{attribute 'TcGenerated'}
{attribute 'no-analysis'}
{attribute 'linkalways'}
// This function has been automatically generated from the project information.
VAR_GLOBAL CONSTANT
	{attribute 'const_non_replaced'}
	stLibVersion_Intecre_File : ST_LibVersion := (iMajor := 0, iMinor := 2, iBuild := 0, iRevision := 0, sVersion := '0.2.0');
END_VAR

(* stored: Version 1.1.0.1, ProductVersion 3.1.4022.18
   GVL Global_Version: Id {cd37158a-2e6c-4471-8e06-19fd2c353fbd} *)
